{attribute 'OPC.UA.DA.StructuredType' := '1'}
TYPE STransition :
STRUCT
	// determines whether this transition in a SStrategy's transition array is part of the strategy.
	IsSet: BOOL;
	
	// -1 signifies unset (because ID 0 is the start node)
	PrevStepIds: ARRAY [ResiConst.ARR_MIN..ResiConst.STRAT_PARALLEL_MAX] OF INT;
	// -1 signifies unset (because ID 0 is the start node)	
	NextStepIds: ARRAY [ResiConst.ARR_MIN..ResiConst.STRAT_PARALLEL_MAX] OF INT;
	
	ExpressionType: EExpressionType;
	ExpressionIdx: UINT;
END_STRUCT
END_TYPE

(* stored: Version 1.1.0.1
   DUT STransition: Id {0900d58e-a6e8-433e-a353-ce98bae666fe} *)
